FUNCTION_BLOCK FB_ManualImplementation_1 IMPLEMENTS  I_ManualImplementation
VAR_INPUT
		i_ManualControl : ARRAY[0..10,0..10] OF I_ManualControl;
END_VAR
VAR_OUTPUT
END_VAR
VAR
	i: INT;
	j: INT;
	k: INT;
	k_1: INT;
END_VAR

//=========================================================
// Instantiation Logic


	FOR k:=0 TO 10 DO
		FOR k_1 := 0 TO 10 DO
			IF i_ManualControl[k, k_1] <> 0 THEN
			THIS^.i_ManualControl[k, k_1] := i_ManualControl[k, k_1];
		END_IF	
		END_FOR
		
	END_FOR


//=========================================================
// Count Declaration Logic

	

//=========================================================
// Manual Logic
	
	//Manual Logic for Vessels.Valves
	
	FOR i:=0 TO 8 DO
		FOR j :=0 TO 7 DO
			IO.Vessels[i].Valves[j].Output :=i_ManualControl[i, j].
				M_RunValve(IO.Vessels[i].Valves[j].bStart);
		END_FOR
	END_FOR
	
	//Manual Logic for Vessels.Pumps
	
	FOR i:=0 TO 8 DO
		FOR j :=0 TO 1 DO
			IO.Vessels[i].Pumps[j].nPulse := 4;
			IO.Vessels[i].Pumps[j].Output :=i_ManualControl[i,j].
				M_RunPump(IO.Vessels[i].Pumps[j].bStart,IO.Vessels[i].Pumps[j].nPulse);
		END_FOR
	END_FOR
	
	//Manual Logic for Reactors.Valves
	
	FOR i:=0 TO 1 DO
		FOR j :=0 TO 7 DO
			IO.Reactors[i].Valves[j].Output :=i_ManualControl[9+i,j].
				M_RunValve(IO.Reactors[i].Valves[j].bStart);
		END_FOR
	END_FOR
	
	//Manual Logic for Reactors.Pumps
	
	FOR i:=0 TO 1 DO
		FOR j :=0 TO 1 DO
			IO.Reactors[i].Pumps[j].nPulse := 4;
			IO.Reactors[i].Pumps[j].Output :=i_ManualControl[9+i,j].
				M_RunPump(IO.Reactors[i].Pumps[j].bStart,IO.Reactors[i].Pumps[j].nPulse);
		END_FOR
	END_FOR

PROPERTY ipManualControl : ARRAY [0..10,0..10] OF I_ManualControl
GET
ipManualControl	:= i_ManualControl;
END_GET
END_PROPERTY

END_FUNCTION_BLOCK

(* stored: Version 1.1.0.1, ProductVersion 3.1.4024.5
   POU FB_ManualImplementation_1: Id {31af0994-073f-4722-92d3-d209ed2dc2fa}, SpecialFunc None
   Property ipManualControl: Id {77789584-0b1f-476b-88c6-131d0cd0edb5}
   Get Get: Id {08c888ae-5b5c-4530-b33f-2f9d7f9e95a4} *)
